// TIA Portal V20 export
TYPE "LER_typePartData"
// stored: Access Published
   STRUCT
      ProcessDataRecord : "LER_typeProcessDataRecord";
      Common : "LER_typeCommonData";
      UnitData : "LER_typeUnitResultData";
   END_STRUCT;
END_TYPE
